% RSLogix 500 project Control_VFD.RSS, saved by version 8.30.00.16 %
PROJECT "UNTITLED"    % processor: Bul.1763 MicroLogix 1100 Series B %

PROGRAM FILES
  LAD 2 "MAIN"  4 rungs
  LAD 3 "CONTROLE"  12 rungs

DATA FILES
  O0 OUTPUT  4 elements
  I1 INPUT  6 elements
  S2 STATUS  66 elements
  B3 BINARY  1 elements
  T4 TIMER  1 elements
  C5 COUNTER  1 elements
  R6 CONTROL  1 elements
  N7 INTEGER  6 elements
  F8 FLOAT  3 elements

LADDER 2 "MAIN"
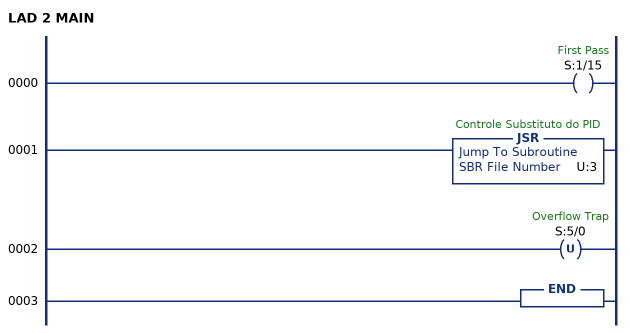
% Rung: 0 %
SOR OTE S:1/15 EOR
%   S:1/15  "First Pass" %
% Rung: 1 %
SOR JSR U:3 EOR
%   U:3  "Controle Substituto do PID" %
% Rung: 2 %
SOR OTU S:5/0 EOR
%   S:5/0  "Overflow Trap" %
% Rung: 3 %
SOR END EOR

LADDER 3 "CONTROLE"
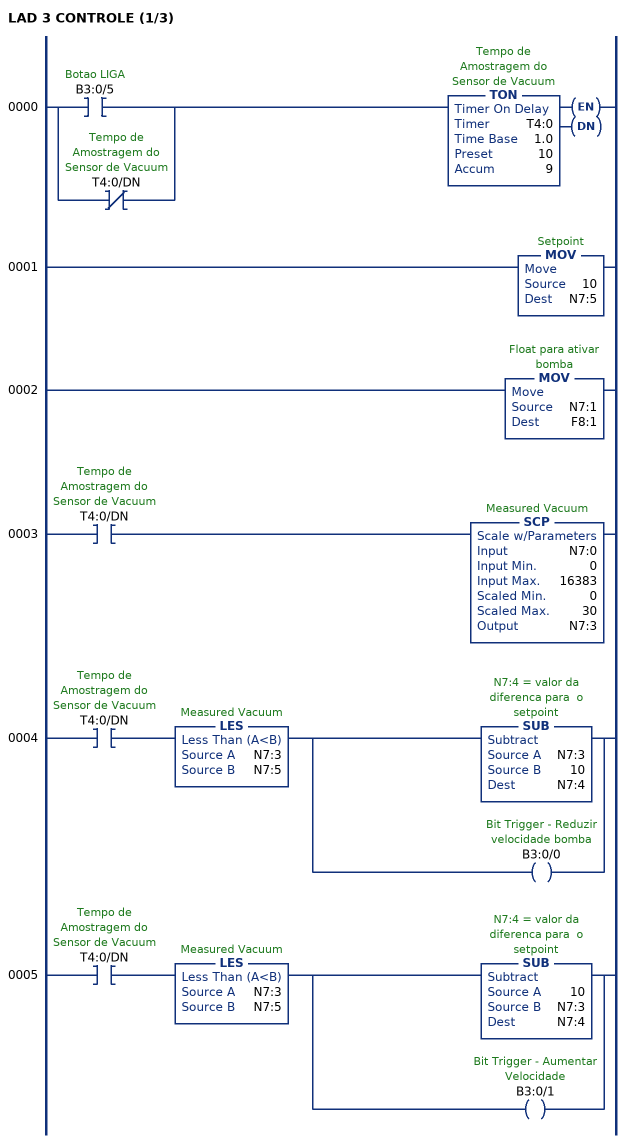
% Rung: 0 %
SOR BST XIC B3:0/5 NXB XIO T4:0/DN BND TON T4:0 1.0 10 9 EOR
%   B3:0/5  "Botao LIGA" %
%   T4:0  "Tempo de Amostragem do Sensor de Vacuum" %
% Rung: 1 %
SOR MOV 10 N7:5 EOR
%   N7:5  "Setpoint" %
% Rung: 2 %
SOR MOV N7:1 F8:1 EOR
%   N7:1  "Vacuum Pump Out" %
%   F8:1  "Float para ativar bomba" %
% Rung: 3 %
SOR XIC T4:0/DN SCP N7:0 0 16383 0 30 N7:3 EOR
%   T4:0  "Tempo de Amostragem do Sensor de Vacuum" %
%   N7:0  "Vacuum sensor in" %
%   N7:3  "Measured Vacuum" %
% Rung: 4 %
SOR XIC T4:0/DN LES N7:3 N7:5 BST SUB N7:3 10 N7:4 NXB OTE B3:0/0 BND EOR
%   T4:0  "Tempo de Amostragem do Sensor de Vacuum" %
%   N7:3  "Measured Vacuum" %
%   N7:5  "Setpoint" %
%   N7:4  "N7:4 = valor da diferenca para  o setpoint" %
%   B3:0/0  "Bit Trigger - Reduzir velocidade bomba" %
% Rung: 5 %
SOR XIC T4:0/DN LES N7:3 N7:5 BST SUB 10 N7:3 N7:4 NXB OTE B3:0/1 BND EOR
%   T4:0  "Tempo de Amostragem do Sensor de Vacuum" %
%   N7:3  "Measured Vacuum" %
%   N7:5  "Setpoint" %
%   N7:4  "N7:4 = valor da diferenca para  o setpoint" %
%   B3:0/1  "Bit Trigger - Aumentar Velocidade" %

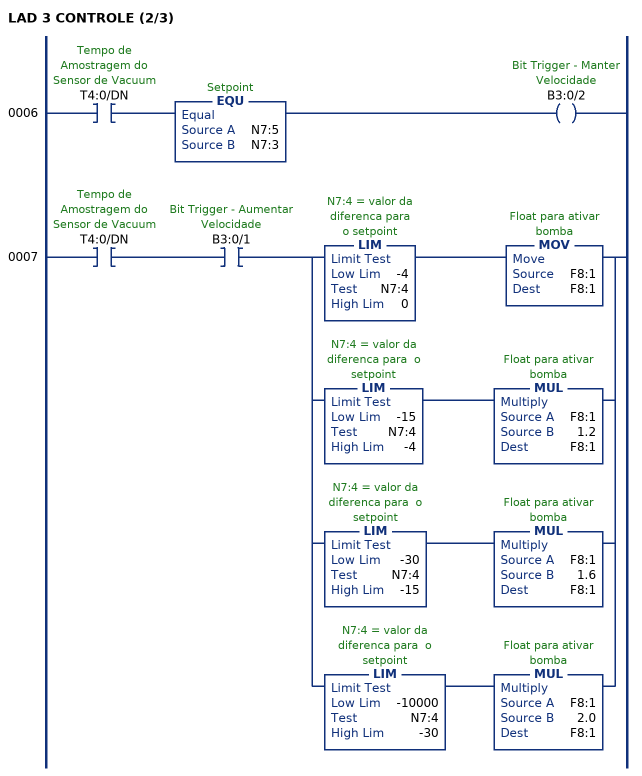
% Rung: 6 %
SOR XIC T4:0/DN EQU N7:5 N7:3 OTE B3:0/2 EOR
%   T4:0  "Tempo de Amostragem do Sensor de Vacuum" %
%   N7:5  "Setpoint" %
%   N7:3  "Measured Vacuum" %
%   B3:0/2  "Bit Trigger - Manter Velocidade" %
% Rung: 7 %
SOR XIC T4:0/DN XIC B3:0/1 BST LIM -4 N7:4 0 MOV F8:1 F8:1 NXB LIM -15 N7:4 -4 MUL F8:1 1.2 F8:1 NXB LIM -30 N7:4 -15 MUL F8:1 1.6 F8:1 NXB LIM -10000 N7:4 -30 MUL F8:1 2.0 F8:1 BND EOR
%   T4:0  "Tempo de Amostragem do Sensor de Vacuum" %
%   B3:0/1  "Bit Trigger - Aumentar Velocidade" %
%   N7:4  "N7:4 = valor da diferenca para  o setpoint" %
%   F8:1  "Float para ativar bomba" %

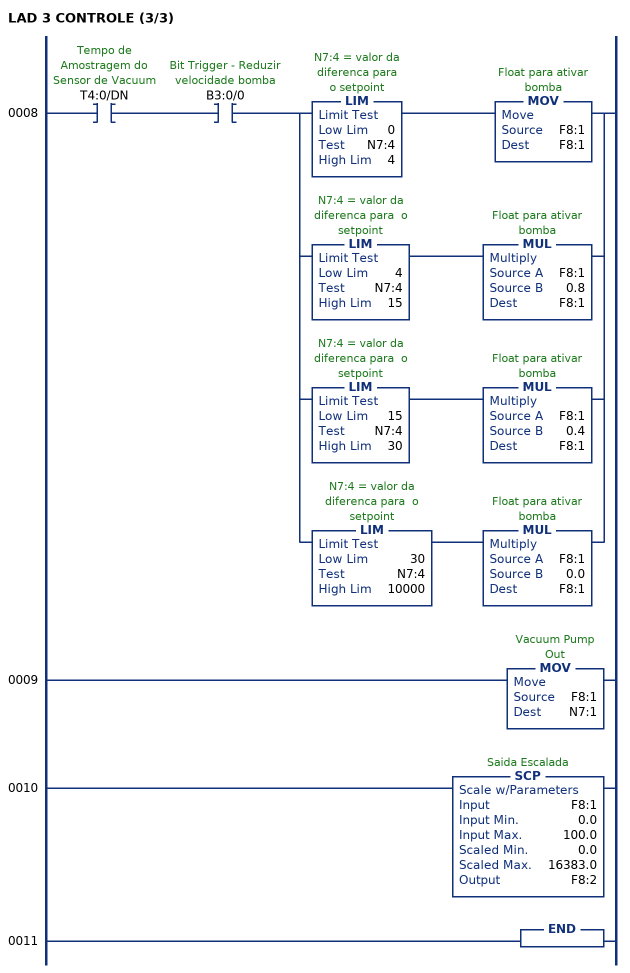
% Rung: 8 %
SOR XIC T4:0/DN XIC B3:0/0 BST LIM 0 N7:4 4 MOV F8:1 F8:1 NXB LIM 4 N7:4 15 MUL F8:1 0.8 F8:1 NXB LIM 15 N7:4 30 MUL F8:1 0.4 F8:1 NXB LIM 30 N7:4 10000 MUL F8:1 0.0 F8:1 BND EOR
%   T4:0  "Tempo de Amostragem do Sensor de Vacuum" %
%   B3:0/0  "Bit Trigger - Reduzir velocidade bomba" %
%   N7:4  "N7:4 = valor da diferenca para  o setpoint" %
%   F8:1  "Float para ativar bomba" %
% Rung: 9 %
SOR MOV F8:1 N7:1 EOR
%   F8:1  "Float para ativar bomba" %
%   N7:1  "Vacuum Pump Out" %
% Rung: 10 %
SOR SCP F8:1 0.0 100.0 0.0 16383.0 F8:2 EOR
%   F8:1  "Float para ativar bomba" %
%   F8:2  "Saida Escalada" %
% Rung: 11 %
SOR END EOR

OTHER DOCUMENTED ADDRESSES
  T4:0/EN  "Trigger Timer"

DATA TABLE (non-zero values as saved)
DATA T4
% .PRE .ACC %
% T4:0 % 10 9
DATA N7
% N7:0 % 3000 3840 0 5 5 10
DATA F8
% F8:0 % 0 3840 629107.2
